// TIA Portal V18 export
VAR_GLOBAL   // PLC tag table "14_SC1-ECL"
   "iSC1-ECL" AT %I8.7 : Bool;
   "oSC1-ECL" AT %Q8.2 : Bool;
END_VAR
